{region '#Template'}
	{attribute 'Category' := 'General'}
	{attribute 'Version' := '0.0.1.0'}
	{attribute 'Tags' := 'General, Building, Operating mode'}
	{attribute 'Description' := 'Gebäude Betriebsart	// Building operating mode'}
{endregion}
FUNCTION_BLOCK FB_BA_BuildingMode EXTENDS FB_BA_View
VAR_INPUT CONSTANT
	OpModMan					: FB_BA_MV_Op;
	OpModPr						: FB_BA_MV_Op;
	Sched						: FB_BA_SchedM;
END_VAR
VAR	
	DeMuxManMod					: FB_BA_DMUX_B04;		
	DeMuxSched					: FB_BA_DMUX_B04;		
	PrioSwi						: FB_BA_PrioSwi_UDI08;	
	
	eBuildingMode				: E_BA_BuildingMode;
	BuildingMode				: FB_BA_RawPublisher;
END_VAR

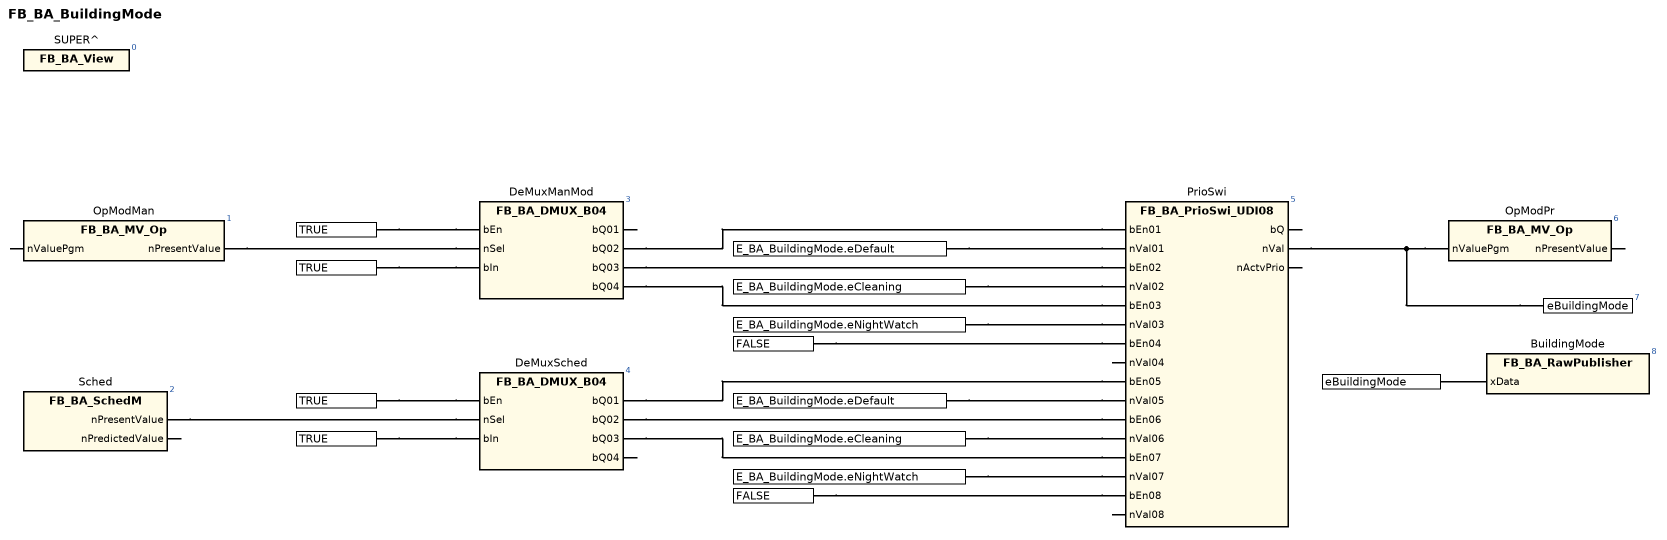
SUPER^(); // FB_BA_View
OpModMan(); // FB_BA_MV_Op
Sched(); // FB_BA_SchedM
DeMuxManMod(bEn := TRUE, nSel := OpModMan.nPresentValue, bIn := TRUE); // FB_BA_DMUX_B04
DeMuxSched(bEn := TRUE, nSel := Sched.nPresentValue, bIn := TRUE); // FB_BA_DMUX_B04
PrioSwi(
    bEn01 := DeMuxManMod.bQ02,
    nVal01 := E_BA_BuildingMode.eDefault,
    bEn02 := DeMuxManMod.bQ03,
    nVal02 := E_BA_BuildingMode.eCleaning,
    bEn03 := DeMuxManMod.bQ04,
    nVal03 := E_BA_BuildingMode.eNightWatch,
    bEn04 := FALSE,
    bEn05 := DeMuxSched.bQ01,
    nVal05 := E_BA_BuildingMode.eDefault,
    bEn06 := DeMuxSched.bQ02,
    nVal06 := E_BA_BuildingMode.eCleaning,
    bEn07 := DeMuxSched.bQ03,
    nVal07 := E_BA_BuildingMode.eNightWatch,
    bEn08 := FALSE); // FB_BA_PrioSwi_UDI08
OpModPr(nValuePgm := PrioSwi.nVal); // FB_BA_MV_Op
eBuildingMode := PrioSwi.nVal;
BuildingMode(xData := eBuildingMode); // FB_BA_RawPublisher

METHOD FB_init : BOOL
VAR_INPUT
	bInitRetains : BOOL; // if TRUE, the retain variables are initialized (warm start / cold start)
	bInCopyCode : BOOL;  // if TRUE, the instance afterwards gets moved into the copy code (online change)
END_VAR
OpModMan.iParent		:= THIS^;	
OpModMan.iLabel			:= LblCmpGeneral.BuildingMode_OpModMan;									
OpModMan.sObjectName	:= '{Idx=01}';
OpModMan.aStateText[1]	:= Texts.txtAuto;
OpModMan.aStateText[2]	:= Texts.txtDefault;
OpModMan.aStateText[3]	:= Texts.txtCleaning;
OpModMan.aStateText[4]	:= Texts.txtNightwatch;
OpModMan.nValueRm		:= 1;

OpModPr.iParent			:= THIS^;	
OpModPr.iLabel			:= LblCmpGeneral.BuildingMode_OpModPr;									
OpModPr.sObjectName		:= '{Idx=01}';
OpModPr.aStateText[1]	:= Texts.txtDefault;
OpModPr.aStateText[2]	:= Texts.txtCleaning;
OpModPr.aStateText[3]	:= Texts.txtNightwatch;
OpModPr.nValueRm		:= 1; 		
                        
Sched.iParent			:= THIS^;	
Sched.iLabel			:= LblCmpGeneral.BuildingMode_Sched;									
Sched.sObjectName		:= '{Idx=01}';
Sched.aStateText[1]		:= Texts.txtDefault;
Sched.aStateText[2]		:= Texts.txtCleaning;
Sched.aStateText[3]		:= Texts.txtNightwatch;
Sched.nPredictTime		:= 0;


Sched.aWeek		:= F_BA_SchedWeekly3xM(E_BA_WeekDay.eMonday, E_BA_WeekDay.eFriday, T#19H, E_BA_BuildingMode.eCleaning, T#20H, E_BA_BuildingMode.eNightWatch, T#6H, E_BA_BuildingMode.eDefault);
(* alternatively
Sched.nDefaultValue										:= E_BA_BuildingMode.eDefault;
Sched.bWriteWeekly										:= FALSE;
//	Monday
Sched.aWeek[E_BA_Weekday.eMonday,1].eState				:= E_BA_SchedEntryState.eValue;
Sched.aWeek[E_BA_Weekday.eMonday,1].uValue.udiVal		:= E_BA_BuildingMode.eCleaning;
Sched.aWeek[E_BA_Weekday.eMonday,1].stTime.nHour		:= 19;
Sched.aWeek[E_BA_Weekday.eMonday,1].stTime.nMinute		:= 0;
Sched.aWeek[E_BA_Weekday.eMonday,1].stTime.nSecond		:= 0;
Sched.aWeek[E_BA_Weekday.eMonday,2].eState				:= E_BA_SchedEntryState.eValue;
Sched.aWeek[E_BA_Weekday.eMonday,2].uValue.udiVal		:= E_BA_BuildingMode.eNightWatch;
Sched.aWeek[E_BA_Weekday.eMonday,2].stTime.nHour		:= 20;
Sched.aWeek[E_BA_Weekday.eMonday,2].stTime.nMinute		:= 0;
Sched.aWeek[E_BA_Weekday.eMonday,2].stTime.nSecond		:= 0;
Sched.aWeek[E_BA_Weekday.eMonday,3].eState				:= E_BA_SchedEntryState.eValue;
Sched.aWeek[E_BA_Weekday.eMonday,3].uValue.udiVal		:= E_BA_BuildingMode.eDefault;
Sched.aWeek[E_BA_Weekday.eMonday,3].stTime.nHour		:= 0;
Sched.aWeek[E_BA_Weekday.eMonday,3].stTime.nMinute		:= 0;
Sched.aWeek[E_BA_Weekday.eMonday,3].stTime.nSecond		:= 0;
//	Tuesday
Sched.aWeek[E_BA_Weekday.eTuesday,1].eState				:= E_BA_SchedEntryState.eValue;
Sched.aWeek[E_BA_Weekday.eTuesday,1].uValue.udiVal		:= E_BA_BuildingMode.eCleaning;
Sched.aWeek[E_BA_Weekday.eTuesday,1].stTime.nHour		:= 19;
Sched.aWeek[E_BA_Weekday.eTuesday,1].stTime.nMinute		:= 0;
Sched.aWeek[E_BA_Weekday.eTuesday,1].stTime.nSecond		:= 0;
Sched.aWeek[E_BA_Weekday.eTuesday,2].eState				:= E_BA_SchedEntryState.eValue;
Sched.aWeek[E_BA_Weekday.eTuesday,2].uValue.udiVal		:= E_BA_BuildingMode.eNightWatch;
Sched.aWeek[E_BA_Weekday.eTuesday,2].stTime.nHour		:= 20;
Sched.aWeek[E_BA_Weekday.eTuesday,2].stTime.nMinute		:= 0;
Sched.aWeek[E_BA_Weekday.eTuesday,2].stTime.nSecond		:= 0;
Sched.aWeek[E_BA_Weekday.eTuesday,3].eState				:= E_BA_SchedEntryState.eValue;
Sched.aWeek[E_BA_Weekday.eTuesday,3].uValue.udiVal		:= E_BA_BuildingMode.eDefault;
Sched.aWeek[E_BA_Weekday.eTuesday,3].stTime.nHour		:= 0;
Sched.aWeek[E_BA_Weekday.eTuesday,3].stTime.nMinute		:= 0;
Sched.aWeek[E_BA_Weekday.eTuesday,3].stTime.nSecond		:= 0;
//	Wednesday
Sched.aWeek[E_BA_Weekday.eWednesday,1].eState			:= E_BA_SchedEntryState.eValue;
Sched.aWeek[E_BA_Weekday.eWednesday,1].uValue.udiVal	:= E_BA_BuildingMode.eCleaning;
Sched.aWeek[E_BA_Weekday.eWednesday,1].stTime.nHour		:= 19;
Sched.aWeek[E_BA_Weekday.eWednesday,1].stTime.nMinute	:= 0;
Sched.aWeek[E_BA_Weekday.eWednesday,1].stTime.nSecond	:= 0;
Sched.aWeek[E_BA_Weekday.eWednesday,2].eState			:= E_BA_SchedEntryState.eValue;
Sched.aWeek[E_BA_Weekday.eWednesday,2].uValue.udiVal	:= E_BA_BuildingMode.eNightWatch;
Sched.aWeek[E_BA_Weekday.eWednesday,2].stTime.nHour		:= 20;
Sched.aWeek[E_BA_Weekday.eWednesday,2].stTime.nMinute	:= 0;
Sched.aWeek[E_BA_Weekday.eWednesday,2].stTime.nSecond	:= 0;
Sched.aWeek[E_BA_Weekday.eWednesday,3].eState			:= E_BA_SchedEntryState.eValue;
Sched.aWeek[E_BA_Weekday.eWednesday,3].uValue.udiVal	:= E_BA_BuildingMode.eDefault;
Sched.aWeek[E_BA_Weekday.eWednesday,3].stTime.nHour		:= 0;
Sched.aWeek[E_BA_Weekday.eWednesday,3].stTime.nMinute	:= 0;
Sched.aWeek[E_BA_Weekday.eWednesday,3].stTime.nSecond	:= 0;
//	Thursday
Sched.aWeek[E_BA_Weekday.eThursday,1].eState			:= E_BA_SchedEntryState.eValue;
Sched.aWeek[E_BA_Weekday.eThursday,1].uValue.udiVal		:=E_BA_BuildingMode.eCleaning;
Sched.aWeek[E_BA_Weekday.eThursday,1].stTime.nHour		:= 19;
Sched.aWeek[E_BA_Weekday.eThursday,1].stTime.nMinute	:= 0;
Sched.aWeek[E_BA_Weekday.eThursday,1].stTime.nSecond	:= 0;
Sched.aWeek[E_BA_Weekday.eThursday,2].eState			:= E_BA_SchedEntryState.eValue;
Sched.aWeek[E_BA_Weekday.eThursday,2].uValue.udiVal		:= E_BA_BuildingMode.eNightWatch;
Sched.aWeek[E_BA_Weekday.eThursday,2].stTime.nHour		:= 20;
Sched.aWeek[E_BA_Weekday.eThursday,2].stTime.nMinute	:= 0;
Sched.aWeek[E_BA_Weekday.eThursday,2].stTime.nSecond	:= 0;
Sched.aWeek[E_BA_Weekday.eThursday,3].eState			:= E_BA_SchedEntryState.eValue;
Sched.aWeek[E_BA_Weekday.eThursday,3].uValue.udiVal		:= E_BA_BuildingMode.eDefault;
Sched.aWeek[E_BA_Weekday.eThursday,3].stTime.nHour		:= 0;
Sched.aWeek[E_BA_Weekday.eThursday,3].stTime.nMinute	:= 0;
Sched.aWeek[E_BA_Weekday.eThursday,3].stTime.nSecond	:= 0;
//	Friday
Sched.aWeek[E_BA_Weekday.eFriday,1].eState				:= E_BA_SchedEntryState.eValue;
Sched.aWeek[E_BA_Weekday.eFriday,1].uValue.udiVal		:= E_BA_BuildingMode.eCleaning;
Sched.aWeek[E_BA_Weekday.eFriday,1].stTime.nHour		:= 19;
Sched.aWeek[E_BA_Weekday.eFriday,1].stTime.nMinute		:= 0;
Sched.aWeek[E_BA_Weekday.eFriday,1].stTime.nSecond		:= 0;
Sched.aWeek[E_BA_Weekday.eFriday,2].eState				:= E_BA_SchedEntryState.eValue;
Sched.aWeek[E_BA_Weekday.eFriday,2].uValue.udiVal		:= E_BA_BuildingMode.eNightWatch;
Sched.aWeek[E_BA_Weekday.eFriday,2].stTime.nHour		:= 20;
Sched.aWeek[E_BA_Weekday.eFriday,2].stTime.nMinute		:= 0;
Sched.aWeek[E_BA_Weekday.eFriday,2].stTime.nSecond		:= 0;
Sched.aWeek[E_BA_Weekday.eFriday,3].eState				:= E_BA_SchedEntryState.eValue;
Sched.aWeek[E_BA_Weekday.eFriday,3].uValue.udiVal		:= E_BA_BuildingMode.eDefault;
Sched.aWeek[E_BA_Weekday.eFriday,3].stTime.nHour		:= 0;
Sched.aWeek[E_BA_Weekday.eFriday,3].stTime.nMinute		:= 0;
Sched.aWeek[E_BA_Weekday.eFriday,3].stTime.nSecond		:= 0; 
*)
END_METHOD

END_FUNCTION_BLOCK

(* stored: Version 1.1.0.1, ProductVersion 3.1.4024.6
   POU FB_BA_BuildingMode: Id {b1acc67f-262e-487d-a42e-5401dce7704e}, SpecialFunc None
   Method FB_init: Id {16a3a86e-b248-4227-825e-772a74d0f2e4} *)
